FUNCTION_BLOCK FB_InternalPowerSupply_IO
VAR
	b_Write					AT %Q* : ARRAY[1..4] OF BOOL;	
	b_Read					AT %I* : ARRAY[1..7] OF BOOL;
END_VAR

VAR_INPUT 
	setACconnectionMode		: BYTE:= 2; // 0: No AC, 1: Grid AC, 2: CEE AC (default)
	b_InternalHVDCConnected : BOOL := FALSE;
	b_DCPsuEnable			: BOOL := FALSE;
	b_ACPsuEnable			: BOOL := TRUE;
	b_KillSupplies			: BOOL := FALSE;
END_VAR

VAR_OUTPUT
	DCPSU_OK: BOOL;
	ACPSU_OK: BOOL;
	GridFuseOK: BOOL;
	CeeFuseOK: BOOL;
	CEE_ACAvailable: BOOL;
	SwitchPSU_OK: BOOL;
	
END_VAR


read();
write();

METHOD GetACconnectionMode : BYTE // 0:= NO ac, 1:= Grid AC, 2:= CEE AC
//IF AC existing give feedback
GetACconnectionMode := 0;
//IF ACPSU_OK THEN
IF b_Write[2] THEN
	GetACconnectionMode := 1;
ELSIF b_Write[1] THEN
	GetACconnectionMode := 2;
END_IF
//END_IF
END_METHOD

METHOD PRIVATE Read : BOOL
VAR
	CEE_ACLeftRotation : BOOL;
	CEE_ACRightRotation: BOOL;
END_VAR
DCPSU_OK := b_read[1];
ACPSU_OK := b_read[2];
GridFuseOK := b_read[3];
CeeFuseOK := b_read[4];
CEE_ACLeftRotation := b_read[5];
CEE_ACRightRotation := b_read[6];
CEE_ACAvailable := CEE_ACLeftRotation OR CEE_ACRightRotation;
SwitchPSU_OK  := b_read[7];
END_METHOD

METHOD Write : BOOL
VAR_INPUT
END_VAR
//B_write[1] = Main supply enable (53Q2)
//B_write[2] = CEE supply enable (53Q1)

IF NOT b_KillSupplies THEN
	// 0: No AC, 1: Grid AC, 2: CEE AC
	CASE setACconnectionMode OF
	0: b_Write[2] := FALSE; b_Write[1] := FALSE;
	1: b_Write[2] := TRUE; 	b_Write[1] := FALSE;
	2: b_Write[2] := FALSE; b_Write[1] := TRUE;
	END_CASE
	
//	IF NOT b_ACPsuEnable THEN
//	b_Write[2] := FALSE; b_Write[1] := FALSE;
//	END_IF
	
	//HVDC disconnect contactors, Only opened in emergency situations when HVDC disconnect fails.
	//Opening these contactors also removes insulation monitor functionality.
	b_Write[3] := b_InternalHVDCConnected;
	b_Write[4] := b_DCPsuEnable;
ELSE
	b_Write[1] := FALSE;
	b_Write[2] := FALSE;
	b_Write[3] := FALSE;
	b_Write[4] := FALSE;
	
END_IF
END_METHOD

END_FUNCTION_BLOCK

(* stored: Version 1.1.0.1, ProductVersion 3.1.4024.12
   POU FB_InternalPowerSupply_IO: Id {14a37718-20e2-4b4a-9114-4d8672574bf3}, SpecialFunc None
   Method GetACconnectionMode: Id {b5d8bdc7-15a4-43f2-8e79-894a816ea164}
   Method Read: Id {3abfc194-ebd1-4f08-a32f-1db20681e61e}
   Method Write: Id {96b4184b-7b1f-4856-9811-3cf26c7cd803} *)
